# EPICS autosave request: apps/xpsMotorApp/Db/hpsTargetScan.req
$(PREF)HPS-XPS:m1:scan1.P1PA
$(PREF)HPS-XPS:m1:scan1.P1SM
$(PREF)HPS-XPS:m1:scan1.P1SP
$(PREF)HPS-XPS:m1:scan1.P1EP
$(PREF)HPS-XPS:m1:scan1.NPTS
$(PREF)HPS-XPS:m1:saveData_scanNumber
$(PREF)HPS-XPS:m1:saveData_fileSystem
$(PREF)HPS-XPS:m1:saveData_subDir
$(PREF)HPS-XPS:m1:saveData_baseName
$(PREF)HPS-XPS:m1:scan1.PDLY
$(PREF)HPS-XPS:m1:scan1.DDLY
